FUNCTION_BLOCK Profile_Velocity_Mode
VAR_INPUT
	NodeID					: BYTE; (* This Port No. addresses the CANopen Node (see System Manager) *)
	Start 					: BOOL;
	Current_State 			: E_Statemachine_State;	
	Statusword				: WORD;	
	Profile_velocity_parameters	: ST_Profile_velocity_parameters;
END_VAR
VAR_OUTPUT
	Controlword 			: WORD;
	Mode_of_operation 		: E_Mode_of_operation	:= E_Mode_of_operation.No_mode_active;
	Target_velocity			: DINT;
	Encoder_offset			: WORD;
	Finished				: BOOL;
END_VAR
VAR
	Index 			: BYTE := 0;
	
	SDO_WRITE		: FB_SDO_WRITE;
	WriteData		: ARRAY [0..255] OF BYTE;
	
	Start_old		: BOOL := FALSE;
END_VAR

// Restart after complete run
IF NOT Start_old AND Start THEN
	Index := 0;
	Finished := FALSE;
END_IF


CASE Index OF	
	0: // Switch to state 'Switch on disabled'
		IF (Start) THEN
			Mode_of_operation := E_Mode_of_operation.No_mode_active;
			Target_velocity	:= 0;	
			Controlword := CONTROLWORD_STATE_CHANGE(Current_State, E_Statemachine_State.Switch_on_disabled);
			IF (Current_State = E_Statemachine_State.Switch_on_disabled) THEN			
				Index := Index + 2;
			ELSE
				Index := Index + 1;		
			END_IF
		END_IF
		
			
	1: // Wait for 'Switch on disabled'
		Controlword := CONTROLWORD_STATE_CHANGE(Current_State, E_Statemachine_State.Switch_on_disabled);	
		IF (Current_State = E_Statemachine_State.Switch_on_disabled) THEN			
			Index := Index + 1;		
		END_IF
		
		
	2: // Set Mode of operation and Acceleration
		Mode_of_operation := E_Mode_of_operation.Profile_velocity_mode;	
		Controlword := CONTROLWORD_STATE_CHANGE(Current_State, E_Statemachine_State.Switch_on_disabled);				
		WriteData[0] := DWORD_TO_BYTE(Profile_velocity_parameters.Profile_acceleration);
		WriteData[1] := DWORD_TO_BYTE(SHR(Profile_velocity_parameters.Profile_acceleration,8));
		WriteData[2] := DWORD_TO_BYTE(SHR(Profile_velocity_parameters.Profile_acceleration,16));
		WriteData[3] := DWORD_TO_BYTE(SHR(Profile_velocity_parameters.Profile_acceleration,24));	
		SDO_WRITE(	
			AdsNetID		:= GLB.ADSNetID_CAN,
			PortNr			:= 16#1000 + GLB.NodeID,
			CO_Index		:= 16#6083,
			CO_SubIndex		:= 16#00,
			DataLength		:= 4,
			WriteData		:= WriteData,
			StartWriting	:= TRUE	
		);	
		Index := Index + 1;		
		
	3: // Wait for finish sdo transfer	
		Controlword := CONTROLWORD_STATE_CHANGE(Current_State, E_Statemachine_State.Switch_on_disabled);	
		SDO_WRITE(StartWriting := FALSE);
		IF SDO_WRITE.WriteDataFinished THEN
			Index := Index + 1;			
		END_IF	
		
		
	4: // Set Deceleration			
		Controlword := CONTROLWORD_STATE_CHANGE(Current_State, E_Statemachine_State.Switch_on_disabled);	
		WriteData[0] := DWORD_TO_BYTE(Profile_velocity_parameters.Profile_deceleration);
		WriteData[1] := DWORD_TO_BYTE(SHR(Profile_velocity_parameters.Profile_deceleration,8));
		WriteData[2] := DWORD_TO_BYTE(SHR(Profile_velocity_parameters.Profile_deceleration,16));
		WriteData[3] := DWORD_TO_BYTE(SHR(Profile_velocity_parameters.Profile_deceleration,24));	
		SDO_WRITE(	
			AdsNetID		:= GLB.ADSNetID_CAN,
			PortNr			:= 16#1000 + GLB.NodeID,
			CO_Index		:= 16#6084,
			CO_SubIndex		:= 16#00,
			DataLength		:= 4,
			WriteData		:= WriteData,
			StartWriting	:= TRUE	
		);	
		Index := Index + 1;		
		
	5: // Wait for finish sdo transfer	
		Controlword := CONTROLWORD_STATE_CHANGE(Current_State, E_Statemachine_State.Switch_on_disabled);	
		SDO_WRITE(StartWriting := FALSE);
		IF SDO_WRITE.WriteDataFinished THEN
			Index := Index + 1;			
		END_IF					
		
	6: // Set  velocity	
		Controlword := CONTROLWORD_STATE_CHANGE(Current_State, E_Statemachine_State.Switch_on_disabled);	
		Target_velocity	:= Profile_velocity_parameters.Target_velocity;
		Index := Index + 1;		
		
	7: // Switch State to 'Operation enabled'
		Controlword := CONTROLWORD_STATE_CHANGE(Current_State, E_Statemachine_State.Operation_enabled);		
		IF (Current_State = E_Statemachine_State.Operation_enabled) THEN			
			Index := 255;
		END_IF
				
		
	255: // Finished 
		FINISHED := TRUE;
				
		
	ELSE
		Index := 255;
			
END_CASE


Start_old := Start;

END_FUNCTION_BLOCK

(* stored: Version 1.1.0.1, ProductVersion 3.1.4024.11
   POU Profile_Velocity_Mode: Id {f383ce37-b1b5-4234-9510-fd3b3ed64452}, SpecialFunc None *)
